# EPICS substitutions: evrSupport/Db/ioc/IOC-LI21-BL01trig.substitutions
# Trigger records
#
# refer to Sharepoint document: Controls | Timing | timingTriggers.xls
#
# Must also have pattern records
# Note: WID, DES, TEC are in terms of nSec and are unique per device
#
file evrDevTrig.db {
#      Device	      , Description   , EVR  ,  width ,desired  , EC delay   , EVR  , EVR,  IOC          , slope
#			                            Trigger       wrt TREF   wrt fiducial loca   unit                 1/119Mhz
  pattern { DEV       ,  DESC         , T    ,  WID   , DES     , TEC        , LOCA , UNIT, IOC          , ESLO
                      ,  PREC         , EGU  ,  DRVL  , DRVH    , EVG}
	  { BLEN:LI21:265:,  "BL11"       , 0    ,  100   , 10      , LCLSBEAM   , LI21 , BL01, IOC:LI21:BL01, 8.40336692324359
                      ,  1            ,"nSec", -2.8E06, 2.8E06  , IN20:EV01}
	  { BLEN:LI21:280:,  "BL12"       , 1    ,  100   , 10      , LCLSBEAM   , LI21 , BL01, IOC:LI21:BL01, 8.40336692324359
                      ,  1            ,"nSec", -2.8E06, 2.8E06  , IN20:EV01}
}
